// TIA Portal V20 export
TYPE "S300ForceMode"
// stored: Access Published, Namespace Global
   STRUCT
      BeltDir : Bool;
      RollerDir : Bool;
   END_STRUCT;
END_TYPE
